FUNCTION_BLOCK SearchEnOcean
VAR_INPUT
END_VAR
VAR_OUTPUT
END_VAR
VAR
	EnOceanSearch: FB_EnOcean_Search;
	byNode: BYTE;
	bReceive: BOOL;
	ar_ID: ARRAY [0..255] OF DWORD;
	iDevices: INT;
END_VAR

//Search and get EnOcean IDs
EnOceanSearch(
	bStart:= TRUE, 
	str_KL6581:= IO.str_KL6581, 
	byNode:= byNode, 
	bReceive=> bReceive, 
	iDevices=> iDevices, 
	ar_ID=> ar_ID);

END_FUNCTION_BLOCK

(* stored: Version 1.1.0.1, ProductVersion 3.1.4022.16
   POU SearchEnOcean: Id {60738440-23f4-493b-aa50-acb6bbcc1b7d}, SpecialFunc None *)
